% RSLogix 500 project main.RSS, saved by version 7.10.00.09 %
PROJECT "SLC05"    % processor: type code 26 %

PROGRAM FILES
  LAD 2 "MAIN"  27 rungs
  LAD 3 "WAHING"  10 rungs
  LAD 4 "RL_W"  9 rungs
  LAD 5 "RR_W"  8 rungs
  LAD 6 "SEP"  9 rungs

DATA FILES
  O0 OUTPUT  11 elements
  I1 INPUT  11 elements
  S2 STATUS  33 elements
  B3 BINARY  9 elements
  T4 TIMER  30 elements
  C5 COUNTER  6 elements
  R6 CONTROL  13 elements
  N7 INTEGER  24 elements
  T9   1 elements

LADDER 2 "MAIN"
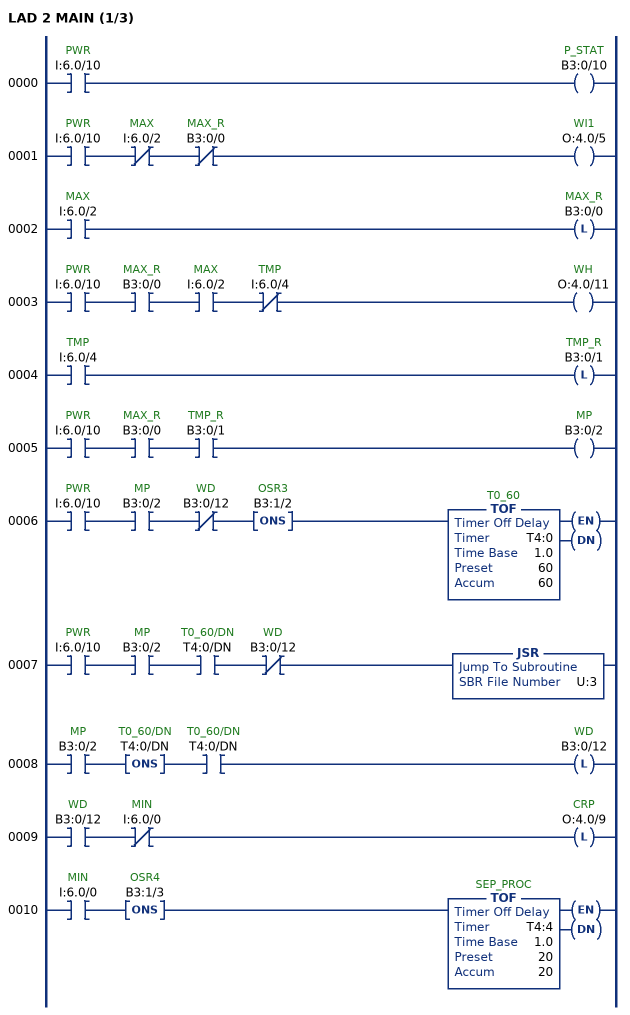
% Rung: 0 %
SOR XIC I:6.0/10 OTE B3:0/10 EOR
%   I:6.0/10  PWR %
%   B3:0/10  P_STAT %
% Rung: 1 %
SOR XIC I:6.0/10 XIO I:6.0/2 XIO B3:0/0 OTE O:4.0/5 EOR
%   I:6.0/10  PWR %
%   I:6.0/2  MAX %
%   B3:0/0  MAX_R %
%   O:4.0/5  WI1 %
% Rung: 2 %
SOR XIC I:6.0/2 OTL B3:0/0 EOR
%   I:6.0/2  MAX %
%   B3:0/0  MAX_R %
% Rung: 3 %
SOR XIC I:6.0/10 XIC B3:0/0 XIC I:6.0/2 XIO I:6.0/4 OTE O:4.0/11 EOR
%   I:6.0/10  PWR %
%   B3:0/0  MAX_R %
%   I:6.0/2  MAX %
%   I:6.0/4  TMP %
%   O:4.0/11  WH %
% Rung: 4 %
SOR XIC I:6.0/4 OTL B3:0/1 EOR
%   I:6.0/4  TMP %
%   B3:0/1  TMP_R %
% Rung: 5 %
SOR XIC I:6.0/10 XIC B3:0/0 XIC B3:0/1 OTE B3:0/2 EOR
%   I:6.0/10  PWR %
%   B3:0/0  MAX_R %
%   B3:0/1  TMP_R %
%   B3:0/2  MP %
% Rung: 6 %
SOR XIC I:6.0/10 XIC B3:0/2 XIO B3:0/12 OSR B3:1/2 TOF T4:0 1.0 60 60 EOR
%   I:6.0/10  PWR %
%   B3:0/2  MP %
%   B3:0/12  WD %
%   B3:1/2  OSR3 %
%   T4:0  T0_60 %
% Rung: 7 %
SOR XIC I:6.0/10 XIC B3:0/2 XIC T4:0/DN XIO B3:0/12 JSR U:3 EOR
%   I:6.0/10  PWR %
%   B3:0/2  MP %
%   T4:0  T0_60 %
%   B3:0/12  WD %
% Rung: 8 %
SOR XIC B3:0/2 OSR T4:0/DN XIC T4:0/DN OTL B3:0/12 EOR
%   B3:0/2  MP %
%   T4:0  T0_60 %
%   B3:0/12  WD %
% Rung: 9 %
SOR XIC B3:0/12 XIO I:6.0/0 OTL O:4.0/9 EOR
%   B3:0/12  WD %
%   I:6.0/0  MIN %
%   O:4.0/9  CRP %
% Rung: 10 %
SOR XIC I:6.0/0 OSR B3:1/3 TOF T4:4 1.0 20 20 EOR
%   I:6.0/0  MIN %
%   B3:1/3  OSR4 %
%   T4:4  SEP_PROC %

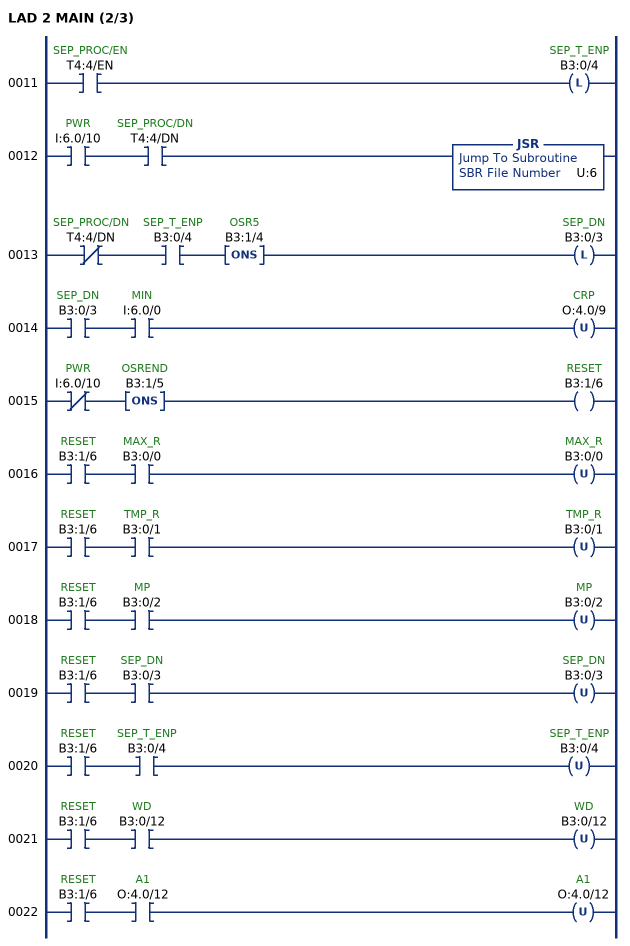
% Rung: 11 %
SOR XIC T4:4/EN OTL B3:0/4 EOR
%   T4:4  SEP_PROC %
%   B3:0/4  SEP_T_ENP %
% Rung: 12 %
SOR XIC I:6.0/10 XIC T4:4/DN JSR U:6 EOR
%   I:6.0/10  PWR %
%   T4:4  SEP_PROC %
% Rung: 13 %
SOR XIO T4:4/DN XIC B3:0/4 OSR B3:1/4 OTL B3:0/3 EOR
%   T4:4  SEP_PROC %
%   B3:0/4  SEP_T_ENP %
%   B3:1/4  OSR5 %
%   B3:0/3  SEP_DN %
% Rung: 14 %
SOR XIC B3:0/3 XIC I:6.0/0 OTU O:4.0/9 EOR
%   B3:0/3  SEP_DN %
%   I:6.0/0  MIN %
%   O:4.0/9  CRP %
% Rung: 15 %
SOR XIO I:6.0/10 OSR B3:1/5 OTE B3:1/6 EOR
%   I:6.0/10  PWR %
%   B3:1/5  OSREND %
%   B3:1/6  RESET %
% Rung: 16 %
SOR XIC B3:1/6 XIC B3:0/0 OTU B3:0/0 EOR
%   B3:1/6  RESET %
%   B3:0/0  MAX_R %
% Rung: 17 %
SOR XIC B3:1/6 XIC B3:0/1 OTU B3:0/1 EOR
%   B3:1/6  RESET %
%   B3:0/1  TMP_R %
% Rung: 18 %
SOR XIC B3:1/6 XIC B3:0/2 OTU B3:0/2 EOR
%   B3:1/6  RESET %
%   B3:0/2  MP %
% Rung: 19 %
SOR XIC B3:1/6 XIC B3:0/3 OTU B3:0/3 EOR
%   B3:1/6  RESET %
%   B3:0/3  SEP_DN %
% Rung: 20 %
SOR XIC B3:1/6 XIC B3:0/4 OTU B3:0/4 EOR
%   B3:1/6  RESET %
%   B3:0/4  SEP_T_ENP %
% Rung: 21 %
SOR XIC B3:1/6 XIC B3:0/12 OTU B3:0/12 EOR
%   B3:1/6  RESET %
%   B3:0/12  WD %
% Rung: 22 %
SOR XIC B3:1/6 XIC O:4.0/12 OTU O:4.0/12 EOR
%   B3:1/6  RESET %
%   O:4.0/12  A1 %

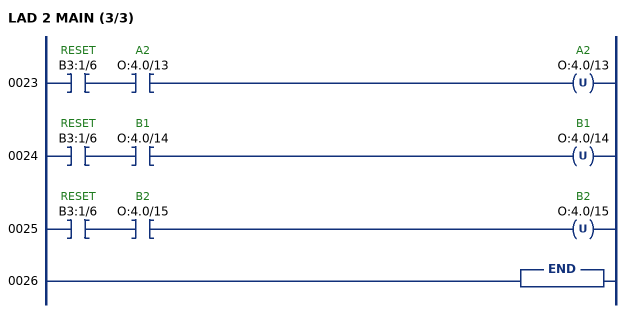
% Rung: 23 %
SOR XIC B3:1/6 XIC O:4.0/13 OTU O:4.0/13 EOR
%   B3:1/6  RESET %
%   O:4.0/13  A2 %
% Rung: 24 %
SOR XIC B3:1/6 XIC O:4.0/14 OTU O:4.0/14 EOR
%   B3:1/6  RESET %
%   O:4.0/14  B1 %
% Rung: 25 %
SOR XIC B3:1/6 XIC O:4.0/15 OTU O:4.0/15 EOR
%   B3:1/6  RESET %
%   O:4.0/15  B2 %
% Rung: 26 %
SOR END EOR

LADDER 3 "WAHING"
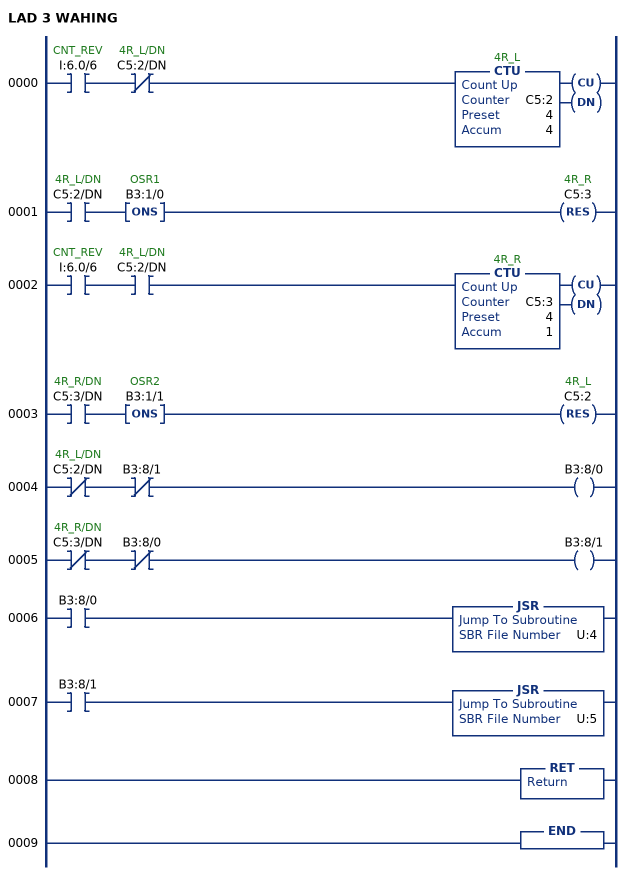
% Rung: 0 %
SOR XIC I:6.0/6 XIO C5:2/DN CTU C5:2 4 4 EOR
%   I:6.0/6  CNT_REV %
%   C5:2  4R_L %
% Rung: 1 %
SOR XIC C5:2/DN OSR B3:1/0 RES C5:3 EOR
%   C5:2  4R_L %
%   B3:1/0  OSR1 %
%   C5:3  4R_R %
% Rung: 2 %
SOR XIC I:6.0/6 XIC C5:2/DN CTU C5:3 4 1 EOR
%   I:6.0/6  CNT_REV %
%   C5:2  4R_L %
%   C5:3  4R_R %
% Rung: 3 %
SOR XIC C5:3/DN OSR B3:1/1 RES C5:2 EOR
%   C5:3  4R_R %
%   B3:1/1  OSR2 %
%   C5:2  4R_L %
% Rung: 4 %
SOR XIO C5:2/DN XIO B3:8/1 OTE B3:8/0 EOR
%   C5:2  4R_L %
% Rung: 5 %
SOR XIO C5:3/DN XIO B3:8/0 OTE B3:8/1 EOR
%   C5:3  4R_R %
% Rung: 6 %
SOR XIC B3:8/0 JSR U:4 EOR
% Rung: 7 %
SOR XIC B3:8/1 JSR U:5 EOR
% Rung: 8 %
SOR RET EOR
% Rung: 9 %
SOR END EOR

LADDER 4 "RL_W"
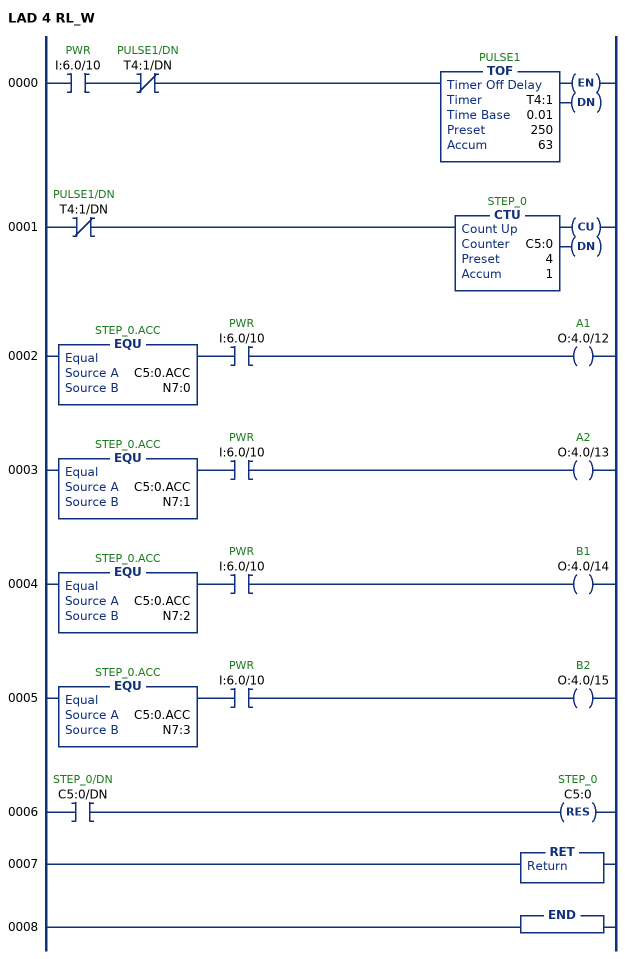
% Rung: 0 %
SOR XIC I:6.0/10 XIO T4:1/DN TOF T4:1 0.01 250 63 EOR
%   I:6.0/10  PWR %
%   T4:1  PULSE1 %
% Rung: 1 %
SOR XIO T4:1/DN CTU C5:0 4 1 EOR
%   T4:1  PULSE1 %
%   C5:0  STEP_0 %
% Rung: 2 %
SOR EQU C5:0.ACC N7:0 XIC I:6.0/10 OTE O:4.0/12 EOR
%   C5:0  STEP_0 %
%   I:6.0/10  PWR %
%   O:4.0/12  A1 %
% Rung: 3 %
SOR EQU C5:0.ACC N7:1 XIC I:6.0/10 OTE O:4.0/13 EOR
%   C5:0  STEP_0 %
%   I:6.0/10  PWR %
%   O:4.0/13  A2 %
% Rung: 4 %
SOR EQU C5:0.ACC N7:2 XIC I:6.0/10 OTE O:4.0/14 EOR
%   C5:0  STEP_0 %
%   I:6.0/10  PWR %
%   O:4.0/14  B1 %
% Rung: 5 %
SOR EQU C5:0.ACC N7:3 XIC I:6.0/10 OTE O:4.0/15 EOR
%   C5:0  STEP_0 %
%   I:6.0/10  PWR %
%   O:4.0/15  B2 %
% Rung: 6 %
SOR XIC C5:0/DN RES C5:0 EOR
%   C5:0  STEP_0 %
% Rung: 7 %
SOR RET EOR
% Rung: 8 %
SOR END EOR

LADDER 5 "RR_W"
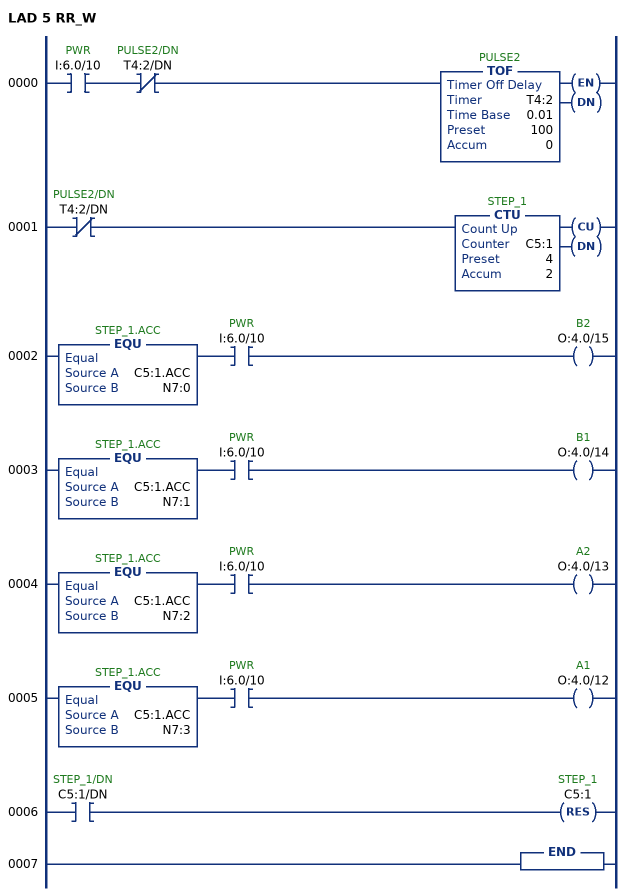
% Rung: 0 %
SOR XIC I:6.0/10 XIO T4:2/DN TOF T4:2 0.01 100 0 EOR
%   I:6.0/10  PWR %
%   T4:2  PULSE2 %
% Rung: 1 %
SOR XIO T4:2/DN CTU C5:1 4 2 EOR
%   T4:2  PULSE2 %
%   C5:1  STEP_1 %
% Rung: 2 %
SOR EQU C5:1.ACC N7:0 XIC I:6.0/10 OTE O:4.0/15 EOR
%   C5:1  STEP_1 %
%   I:6.0/10  PWR %
%   O:4.0/15  B2 %
% Rung: 3 %
SOR EQU C5:1.ACC N7:1 XIC I:6.0/10 OTE O:4.0/14 EOR
%   C5:1  STEP_1 %
%   I:6.0/10  PWR %
%   O:4.0/14  B1 %
% Rung: 4 %
SOR EQU C5:1.ACC N7:2 XIC I:6.0/10 OTE O:4.0/13 EOR
%   C5:1  STEP_1 %
%   I:6.0/10  PWR %
%   O:4.0/13  A2 %
% Rung: 5 %
SOR EQU C5:1.ACC N7:3 XIC I:6.0/10 OTE O:4.0/12 EOR
%   C5:1  STEP_1 %
%   I:6.0/10  PWR %
%   O:4.0/12  A1 %
% Rung: 6 %
SOR XIC C5:1/DN RES C5:1 EOR
%   C5:1  STEP_1 %
% Rung: 7 %
SOR END EOR

LADDER 6 "SEP"
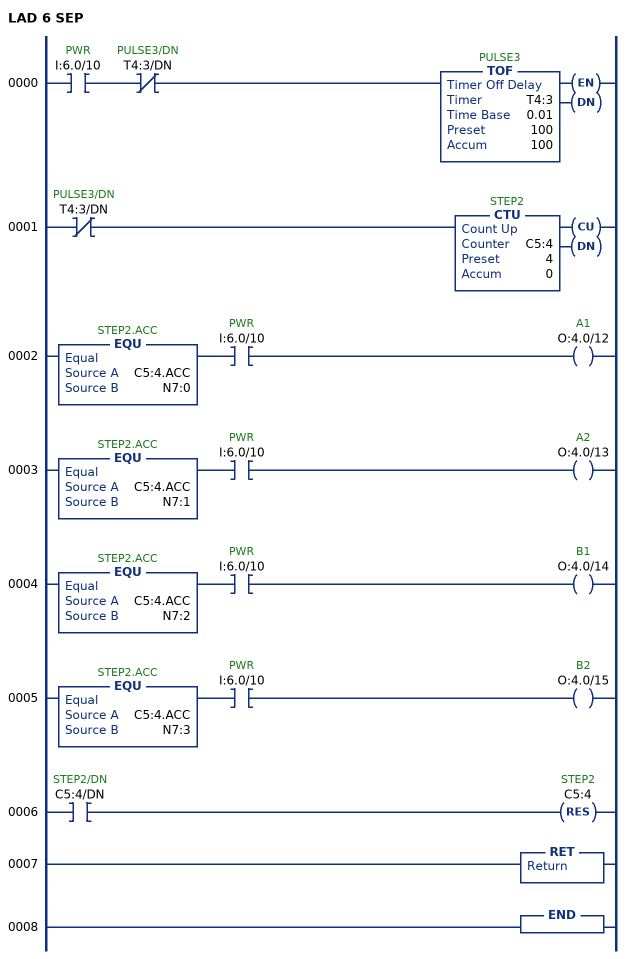
% Rung: 0 %
SOR XIC I:6.0/10 XIO T4:3/DN TOF T4:3 0.01 100 100 EOR
%   I:6.0/10  PWR %
%   T4:3  PULSE3 %
% Rung: 1 %
SOR XIO T4:3/DN CTU C5:4 4 0 EOR
%   T4:3  PULSE3 %
%   C5:4  STEP2 %
% Rung: 2 %
SOR EQU C5:4.ACC N7:0 XIC I:6.0/10 OTE O:4.0/12 EOR
%   C5:4  STEP2 %
%   I:6.0/10  PWR %
%   O:4.0/12  A1 %
% Rung: 3 %
SOR EQU C5:4.ACC N7:1 XIC I:6.0/10 OTE O:4.0/13 EOR
%   C5:4  STEP2 %
%   I:6.0/10  PWR %
%   O:4.0/13  A2 %
% Rung: 4 %
SOR EQU C5:4.ACC N7:2 XIC I:6.0/10 OTE O:4.0/14 EOR
%   C5:4  STEP2 %
%   I:6.0/10  PWR %
%   O:4.0/14  B1 %
% Rung: 5 %
SOR EQU C5:4.ACC N7:3 XIC I:6.0/10 OTE O:4.0/15 EOR
%   C5:4  STEP2 %
%   I:6.0/10  PWR %
%   O:4.0/15  B2 %
% Rung: 6 %
SOR XIC C5:4/DN RES C5:4 EOR
%   C5:4  STEP2 %
% Rung: 7 %
SOR RET EOR
% Rung: 8 %
SOR END EOR

OTHER DOCUMENTED ADDRESSES
  B3:2/0  A1_PREV
  B3:2/1  A2_PREV
  B3:2/2  B1_PREV
  B3:2/3  B2_PREV
  O:4.0/7  WI2
  T4:1/TT  PULSE_1

DATA TABLE (non-zero values as saved)
DATA B3
% B3:0 % 0X0401 0X0002 0X0000 0X0000 0X0000 0X0000 0X0000 0X0000 0X0002
DATA T4
% .PRE .ACC %
% T4:0 % 60 60
% T4:1 % 250 63
% T4:2 % 100 0
% T4:3 % 100 100
% T4:4 % 20 20
% T4:5 % 5 0
% T4:6 % 5 0
% T4:7 % 5 0
% T4:8 % 5 5
% T4:9 % 5 5
% T4:10 % 5 1
% T4:11 % 5 0
% T4:12 % 20 0
% T4:13 % 10 0
% T4:14 % 5 0
% T4:15 % 5 0
% T4:16 % 5 0
% T4:17 % 5 0
DATA C5
% .PRE .ACC %
% C5:0 % 4 1
% C5:1 % 4 2
% C5:2 % 4 4
% C5:3 % 4 1
% C5:4 % 4 0
% C5:5 % 4 4
DATA R6
% .LEN .POS %
% R6:0 % 4 2
% R6:1 % 15 0
% R6:2 % 15 0
% R6:12 % 4 2
DATA N7
% N7:0 % 0 1 2 3 4096 8192 16384 0 0 0
% N7:10 % 0 5 10 15 4096 8192 16384 -32768 0 0
% N7:20 % 0 5 10 15
DATA T9
% .PRE .ACC %
% T9:0 % 5 0
